FUNCTION_BLOCK FB_RoofMotor
VAR_INPUT
	roof_number				: UINT;		// number of roof
	drive_number			: UINT;		// number of drive
	min_position			: INT;		// minimum position of roof
	max_position			: INT;		// maximum position of roof
	real_speed				: INT;		// signed speed
	zero_counter			: BOOL := FALSE;	// reset position counter to zero
	comm					: I_Comm;
	
	// counting filters (insurance; defaults sized from the recordings — plan 2026-08-20)
	counter_debounce		: TIME := T#5MS;	// min. on-time of a sensor pulse. Keep clear of the 10 ms task cycle: at
										// PT = cycle time, ordinary cycle jitter can push the elapsed time on the
										// deciding scan just under PT and drop an otherwise-valid pulse entirely
										// (modelled in testing/check_debounce_aliasing.py). 5 ms sits above the
										// EL1008's ~3 ms input filter and comfortably below one cycle.
	counter_min_spacing		: TIME := T#50MS;	// min. time between accepted counts — keep < rotation period (600 ms)
	
	// stall watchdog
	stall_timeout			: TIME := T#10S;	// max. time moving without an accepted count — keep well above the rotation period (0.6 s at max_speed, slower at min_speed) and the ~3 s until the first count after a start
END_VAR
VAR_OUTPUT PERSISTENT
	position				: INT;	// position
END_VAR
VAR_OUTPUT
	percent_open			: REAL;	// percentage open
	
	// moving
	moving					: BOOL;
	
	// debug: raw (unfiltered, ungated) edge count for validation
	raw_counts				: DINT;
	
	// error 
	motor_error		AT%I*	: BOOL;
	error					: BOOL;
	stall_error				: BOOL;	// moving, but no counter edge for stall_timeout (jammed drive, dead sensor)
	
	// signals from limit switches
	opened			AT%I*	: BOOL;
	closed			AT%I*	: BOOL;
	
	// position on limit switch
	position_open			: INT := -1000;
	position_close			: INT := -1000;
END_VAR
VAR
	// error
	drive_error_event		: FB_EventLog;

	// inductive sensor for counting rotation
	counter			AT%I*	: BOOL;
	counter_trig			: R_TRIG;
	counter_raw_trig		: R_TRIG;	// raw (unfiltered) edge trigger — for validation only
	tonDebounce				: TON;		// level debounce for the sensor pulse
	tonSpacing				: TON;		// rate limit: min. spacing between accepted counts
	tonStall				: TON;		// time since the last accepted count while moving
	bCountAccepted			: BOOL;		// a count was accepted in this cycle
	
	// reset command to drive
	reset_command			: BOOL;
	reset_timer				: TON;
	reset_drive		AT%Q*	: BOOL;
	
	// speed
	speed			AT%Q*	: INT;		// move speed
	direction_open	AT%Q*	: BOOL;		// move direction
	direction_close	AT%Q*	: BOOL;
	
	// position on limit switch
	position_open_on_trig	: R_TRIG;
	position_open_off_trig	: F_TRIG;
	position_close_on_trig	: R_TRIG;
	position_close_off_trig	: F_TRIG;
END_VAR

// signals
error := NOT motor_error;

// reset?
//reset_timer();
IF reset_command THEN
	// set signal and start timer
	reset_drive := TRUE;
	reset_timer(IN := TRUE, PT := T#200MS);
END_IF
IF reset_timer.Q THEN
	// reset everything
	reset_drive := FALSE;
	reset_command := FALSE;
	reset_timer(IN := FALSE);
END_IF

// relative position; FB_Roof still calls the motors with max_position <= min_position when config_error is set,
// and a division by zero stops the user-mode runtime (STATUS_FLOAT_DIVIDE_BY_ZERO)
IF max_position > min_position THEN
	percent_open := 1.0 * (position - min_position) / (max_position - min_position) * 100.0;
ELSE
	percent_open := 0.0;
END_IF

// get direction
direction_open := real_speed > 0;
direction_close := real_speed < 0;

// set moving before the counter gate (motion gate: no counting while idle)
moving := real_speed <> 0;

// counter for position — filtered and gated.
// The limit re-sync in FB_Roof is the primary protection; these layers are
// insurance only. Deliberately NOT gated on the limit switches: that would
// blind the sync check to a broken connection or a stalled drive.
tonDebounce(IN := counter, PT := counter_debounce);	// stable-high filter (kills short glitches)
counter_trig(CLK := tonDebounce.Q);					// edge of the filtered signal

// raw edge count (unfiltered, ungated) — for validation/comparison
counter_raw_trig(CLK := counter);
IF counter_raw_trig.Q THEN
	raw_counts := raw_counts + 1;
END_IF

bCountAccepted := FALSE;
IF counter_trig.Q AND moving THEN					// motion gate
	IF tonSpacing.Q THEN							// spacing window since last accepted count elapsed -> accept
		tonSpacing(IN := FALSE);					// restart the spacing window
		bCountAccepted := TRUE;
		IF direction_open THEN
			position := position + 1;
		ELSIF direction_close THEN
			position := position - 1;
		END_IF
	END_IF
END_IF
tonSpacing(IN := TRUE, PT := counter_min_spacing);	// rate limit timer (runs continuously)

// stall watchdog: driven, but the position counter does not advance (both drives jammed
// gives no position difference, so sync_error cannot see it)
tonStall(IN := moving AND NOT bCountAccepted, PT := stall_timeout);
stall_error := tonStall.Q;

// zero?
IF zero_counter THEN
	position := 0;
	raw_counts := 0;
END_IF

// remember position when entering/leaving limit switches
position_open_on_trig(CLK := opened);
IF position_open_on_trig.Q THEN
	position_open := position;
END_IF
position_open_off_trig(CLK := opened);
IF position_open_off_trig.Q THEN
	position_open := -1000;
END_IF
position_close_on_trig(CLK := closed);
IF position_close_on_trig.Q THEN
	position_close := position;
END_IF
position_close_off_trig(CLK := closed);
IF position_close_off_trig.Q THEN
	position_close := -1000;
END_IF

// absolute speed
speed := ABS(real_speed);

// error
drive_error_event(	
	Trigger 		:= error, 
	Level 			:= ADSLOG_MSGTYPE_ERROR,
	FormatString 	:= 'Drive %s in error state.', 
	OnMessage 		:= CONCAT(CONCAT(CONCAT('#', UINT_TO_STRING(drive_number)), ' of roof #'), UINT_TO_STRING(roof_number)),
	Comm			:= comm);

PROPERTY MovedSinceClosed : INT
GET
IF position_close = -1000 THEN
	MovedSinceClosed := 0;
ELSE
	MovedSinceClosed := ABS(position - position_close);
END_IF
END_GET
END_PROPERTY

PROPERTY MovedSinceOpen : INT
GET
IF position_open = -1000 THEN
	MovedSinceOpen := 0;
ELSE
	MovedSinceOpen := ABS(position - position_open);
END_IF
END_GET
END_PROPERTY

METHOD Reset : BOOL
VAR_INPUT
END_VAR
reset_command := TRUE;
END_METHOD

METHOD SetPosition : BOOL
VAR_INPUT
	position_value		: INT;		// new position value (e.g. min/max_position on limit re-sync)
END_VAR
// 'position' is a VAR_OUTPUT — read-only from outside the FB, so the
// FB_Roof-level limit re-sync sets it through this method.
position := position_value;

// Re-anchor the limit-switch records of a switch that is engaged right now. They hold the counter
// reading at engagement, which is meaningless after the snap (e.g. a restart with the roof half
// open: the switch engages at a wrong reading, the snap then corrects the counter). Left alone,
// MovedSince* would report the correction as travel and raise a false limit_error.
// A drive that really overruns its switch still trips limit_error: that check runs every cycle
// before a snap can happen, and a snap needs both switches engaged.
IF opened THEN
	position_open := position_value;
END_IF
IF closed THEN
	position_close := position_value;
END_IF
END_METHOD

END_FUNCTION_BLOCK

(* stored: Version 1.1.0.1, ProductVersion 3.1.4024.15
   POU FB_RoofMotor: Id {47cefcf1-8ba0-4c06-bdcd-b7d169ce9c61}, SpecialFunc None
   Property MovedSinceClosed: Id {2719aae1-546e-4298-912e-02b6d87518f5}
   Get Get: Id {96f83e28-e8ad-4fde-910b-1a5f42c9fcc0}
   Property MovedSinceOpen: Id {bae22f4e-cf0f-4b68-8c2a-92262cee694d}
   Get Get: Id {86e36bdf-b1ad-4e46-b5a9-f1d0514460ed}
   Method Reset: Id {aa634c66-2ca0-4bfc-8efe-d1b3d9d3132b}
   Method SetPosition: Id {D579E16E-908F-46C7-A5F1-23B0FAF96397} *)
